{attribute 'GeneratedUsingTerminal: KL6224-0003'}
{attribute addProperty BoxType "KL6224-0003"}
{attribute addProperty Id "Channel_1AT %Q*Channel_779103830"}
{attribute addProperty CRC "2126695780"}
{attribute addProperty Size "0"}
TYPE KL_7EC2CD64 :
STRUCT
	{attribute addProperty Name "Channel_1"}
	Channel_1 : Channel_77910383;
END_STRUCT
END_TYPE

(* stored: Version 1.2.0.0, ProductVersion 3.1.4024.9
   DUT KL_7EC2CD64: Id {2595e819-7a40-4179-b326-6884b04f5b05} *)
